FUNCTION WORDS_TO_DWORD
  (* Standard: 61499-1 *)
  (* Version 1.0, 2024-02-22, franz *)
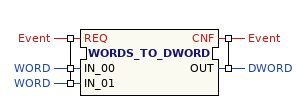
  EVENT_INPUT
    REQ WITH IN_00, IN_01; (* Normal Execution Request *)
  END_EVENT
  EVENT_OUTPUT
    CNF WITH OUT; (* Execution Confirmation *)
  END_EVENT
  VAR_INPUT
    IN_00 : WORD; (* WORD 00 *)
    IN_01 : WORD; (* WORD 01 *)
  END_VAR
  VAR_OUTPUT
    OUT : DWORD; (* DWORD Output *)
  END_VAR
  BODY IN ST:
FUNCTION WORDS_TO_DWORD

VAR_INPUT
	IN_00 : WORD;    // WORD 00
	IN_01 : WORD;    // WORD 01
END_VAR

VAR_OUTPUT
	OUT : DWORD;    // DWORD Output
END_VAR

(* this Function combines the 2 WORDS to a dword *)
OUT := SHL(IN_01, SHIFT_WORD_01)
	OR SHL(IN_00, SHIFT_WORD_00);

END_FUNCTION
  END_BODY
END_FUNCTION
